SYSTEM DRILL_VIEWL (* Drill System View + HMI *)
  (* Standard: 61499-1; Classification: Simulation; ApplicationDomain: Transfer Lines; Function: Drillingd *)
  (* Version 0.1, 2004-10-18, JHC, Rockwell Automation, Changed loader/unloader to SOL_VIEWL. *)
  (* Version 0.0, 2002-04-25, JHC, Rockwell Automation, Adapted from TESTBED_VIEWL *)
  DEVICE HMI : FRAME_DEVICE
    RESOURCE RES1 : PANEL_RESOURCE
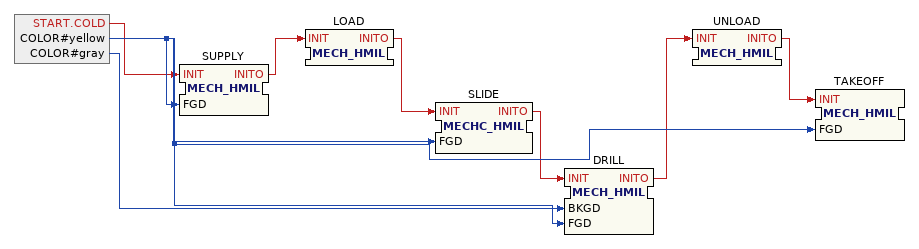
      FBS
        SUPPLY : MECH_HMIL;
        LOAD : MECH_HMIL;
        DRILL : MECH_HMIL;
        SLIDE : MECHC_HMIL;
        UNLOAD : MECH_HMIL;
        TAKEOFF : MECH_HMIL;
      END_FBS
      EVENT_CONNECTIONS
        START.COLD TO SUPPLY.INIT;
        SUPPLY.INITO TO LOAD.INIT;
        LOAD.INITO TO SLIDE.INIT;
        SLIDE.INITO TO DRILL.INIT;
        DRILL.INITO TO UNLOAD.INIT;
        UNLOAD.INITO TO TAKEOFF.INIT;
      END_CONNECTIONS
      DATA_CONNECTIONS
        COLOR#yellow TO SUPPLY.FGD;
        COLOR#yellow TO SLIDE.FGD;
        COLOR#gray TO DRILL.BKGD;
        COLOR#yellow TO DRILL.FGD;
        COLOR#yellow TO TAKEOFF.FGD;
      END_CONNECTIONS
    END_RESOURCE
  END_DEVICE
  DEVICE VIEW : FRAME_DEVICE
    RESOURCE INPUT : VIEW_PANEL
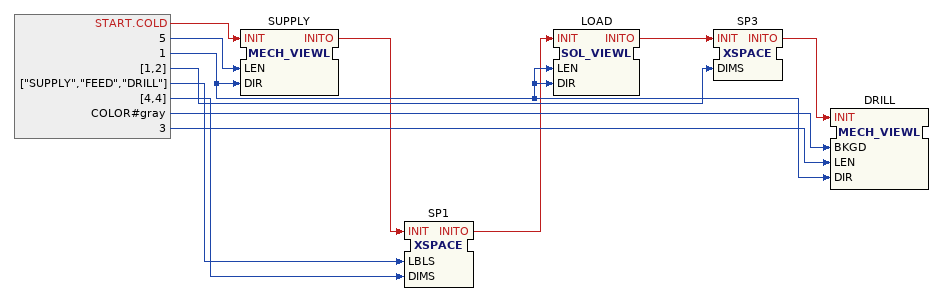
      FBS
        SUPPLY : MECH_VIEWL; (* Supply transfer mechanism *)
        SP1 : XSPACE;
        LOAD : SOL_VIEWL; (* Loader mechanism *)
        SP3 : XSPACE;
        DRILL : MECH_VIEWL;
      END_FBS
      EVENT_CONNECTIONS
        START.COLD TO SUPPLY.INIT;
        SUPPLY.INITO TO SP1.INIT;
        SP1.INITO TO LOAD.INIT;
        LOAD.INITO TO SP3.INIT;
        SP3.INITO TO DRILL.INIT;
      END_CONNECTIONS
      DATA_CONNECTIONS
        5 TO SUPPLY.LEN;
        1 TO SUPPLY.DIR;
        [1,2] TO SP3.DIMS;
        ["SUPPLY","FEED","DRILL"] TO SP1.LBLS;
        [4,4] TO SP1.DIMS;
        COLOR#gray TO DRILL.BKGD;
        3 TO DRILL.LEN;
        1 TO DRILL.DIR;
        1 TO LOAD.LEN;
        1 TO LOAD.DIR;
      END_CONNECTIONS
    END_RESOURCE
    RESOURCE OUTPUT : VIEW_PANEL
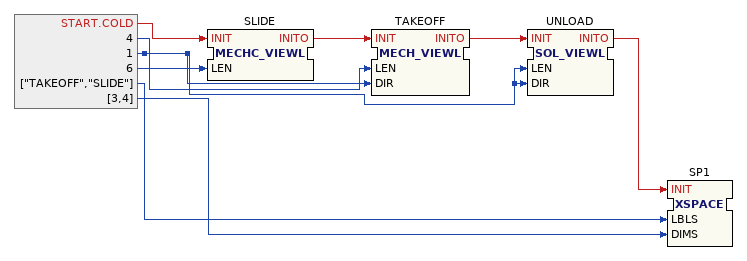
      FBS
        SLIDE : MECHC_VIEWL;
        TAKEOFF : MECH_VIEWL; (* Takeoff Transfer *)
        UNLOAD : SOL_VIEWL; (* Unloader Mechanism *)
        SP1 : XSPACE;
      END_FBS
      EVENT_CONNECTIONS
        START.COLD TO SLIDE.INIT;
        SLIDE.INITO TO TAKEOFF.INIT;
        TAKEOFF.INITO TO UNLOAD.INIT;
        UNLOAD.INITO TO SP1.INIT;
      END_CONNECTIONS
      DATA_CONNECTIONS
        4 TO TAKEOFF.LEN;
        1 TO TAKEOFF.DIR;
        6 TO SLIDE.LEN;
        ["TAKEOFF","SLIDE"] TO SP1.LBLS;
        [3,4] TO SP1.DIMS;
        1 TO UNLOAD.LEN;
        1 TO UNLOAD.DIR;
      END_CONNECTIONS
    END_RESOURCE
    DATA_CONNECTIONS
      0 TO INPUT.TRACE;
      25 TO INPUT.DIA;
      [6,5] TO INPUT.SIZE;
      1 TO INPUT.VERTICAL;
      25 TO OUTPUT.DIA;
      [6,5] TO OUTPUT.SIZE;
    END_CONNECTIONS
  END_DEVICE
  DATA_CONNECTIONS (* parameter values *)
    [100,100,375,200] TO HMI.BOUNDS;
    [1,1] TO HMI.GRID;
    [475,100,220,300] TO VIEW.BOUNDS;
  END_CONNECTIONS
END_SYSTEM
